// Mitsubishi GX Works2 project: 서보   PLC: Q03UDV

PROGRAM MAIN
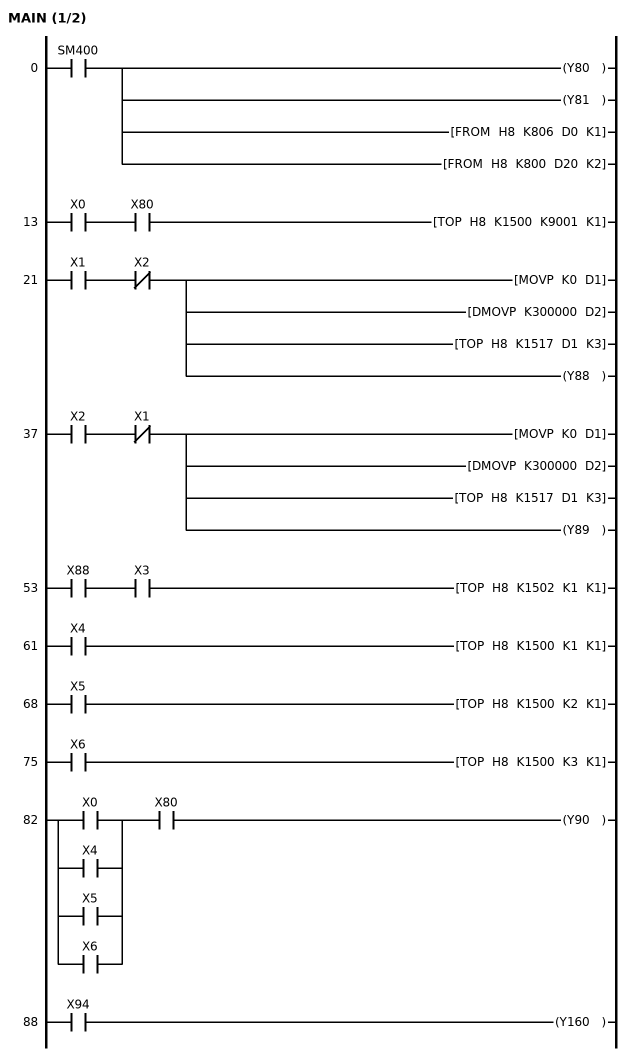
0     LD      SM400
      OUT     Y80
      OUT     Y81
      FROM    H8 K806 D0 K1
      FROM    H8 K800 D20 K2
13    LD      X0
      AND     X80
      TOP     H8 K1500 K9001 K1
21    LD      X1
      ANI     X2
      MOVP    K0 D1
      DMOVP   K300000 D2
      TOP     H8 K1517 D1 K3
      OUT     Y88
37    LD      X2
      ANI     X1
      MOVP    K0 D1
      DMOVP   K300000 D2
      TOP     H8 K1517 D1 K3
      OUT     Y89
53    LD      X88
      AND     X3
      TOP     H8 K1502 K1 K1
61    LD      X4
      TOP     H8 K1500 K1 K1
68    LD      X5
      TOP     H8 K1500 K2 K1
75    LD      X6
      TOP     H8 K1500 K3 K1
82    LD      X0
      OR      X4
      OR      X5
      OR      X6
      AND     X80
      OUT     Y90
88    LD      X94
      OUT     Y160
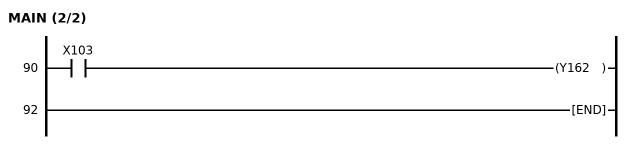
90    LD      X103
      OUT     Y162
92    END
END_PROGRAM
